(* Logix 5000 project; controller R5_CSS vendor 1 type 14 code 74 rev 19.11; software revision 19.01; part 9 of 20 *)
(* tags used below, declared in another part *)
   AC102A_BLEED_MAKEUP_STATUS : DINT;   // 0=stopped 1=bleed water 2=makeup water 3=wait
   AC102A_BLEED_START_TON : TIMER;
   AlarmMaster : DINT;
   F1_LC302 : LEVEL_CONTROL;
   F1_LC303A : LEVEL_CONTROL;
   F1_LC370 : LEVEL_CONTROL;
   FC365_LC370_FLOW_AUTO_SP : REAL;
   FC365_MAX_TIME_MIN : DINT;
   FC370 : FLOW_CONTROL;   // COALESCER MAKE UP WATER FLOW CONTROL
   FC370_FEED_ALARM_DISABLE : BOOL;
   FireFlowAlarmFromUTL : BOOL;
   LC302 : LEVEL_CONTROL;   // COALESCER OIL CHAMBER LEVEL CONTROL
   LC303 : LEVEL_CONTROL;   // COALESCER DIFFEENCE BETWEEN INTERFACE AND AQUEOUS PHASE
   LC303A : LEVEL_CONTROL;   // AQUEOUS PHASE OF PRIMARY SETTLER
   LC303B : LEVEL_CONTROL;   // INTERFACE LEVEL OF PRIMARY CONDENSER
   LC304 : LEVEL_CONTROL;   // SETTLER SECONDARY TANK INTERFACE LEVEL
   LC365_AUTO_SP_START : REAL;
   LC370 : LEVEL_CONTROL;   // WATER MAKE UP FOR PRIMARY SETTLER
   LC370_AUTO_ONS1 : BOOL;
   LC370_AUTO_ONS2 : BOOL;
   LC370_AUTO_SP_START : REAL;
   LC370_Bleed_Makeup_Started : BOOL;
   LC370_FLOW_TOO_LONG_ALM : BOOL;
   LC370_FLOW_TOO_LONG_RESETPB : BOOL;
   LC370_FLOW_TOO_LONG_TMR : TIMER;
   LC370_HMI_MAKEUP_ENABLE : BOOL;
   LC370_HMI_MAKEUP_REQ : BOOL;
   LC370_HMI_MAKEUP_START_ENABLE : BOOL;
   LC370_HMI_MAKEUP_START_PB : BOOL;
   LC370_HMI_MAKEUP_STOP_PB : BOOL;
   LC370_MAKEUP_AUTO_START_TON : TIMER;
   LC370_MANUAL_ONS1 : BOOL;
   LC370_Started : BOOL;
   LC370_TOTAl_GAL : REAL;
   LC370_TOTAl_RESET : BOOL;
   LC370_TOTAl_RESET_PB : BOOL;
   LC370_TOTALIZE : Totalize;
   LC370_TOTALIZE_EN : BOOL;
   LC370_UNABLE_TO_MAKEUP : BOOL;
   PID_LC370_Enable : BOOL;
   PID_LC370_Enable_ONS : BOOL;
   PID_LC370_Enable_Ton : TIMER;
   PID_LCV370 : PID;
   PID_LCV370_TON : TIMER;
   TC313A : TEMP_CONTROL;   // PRIMARY COALESCER SEPARATOR TEMPERATURE CONTROL
   TMR_FAULT : DINT;
(* MainProgram, continued *)

ROUTINE LC302_CoalOilChamberLevel   (* ladder *)
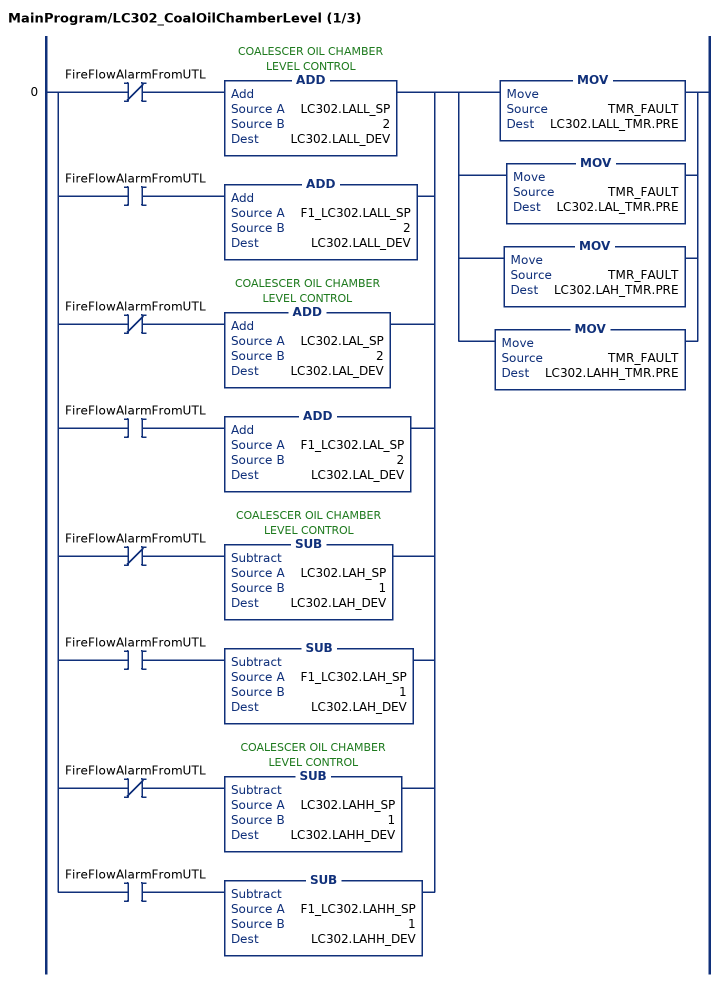
   0: [[XIO(FireFlowAlarmFromUTL) ADD(LC302.LALL_SP,2,LC302.LALL_DEV) ,XIC(FireFlowAlarmFromUTL) ADD(F1_LC302.LALL_SP,2,LC302.LALL_DEV) ] ,[XIO(FireFlowAlarmFromUTL) ADD(LC302.LAL_SP,2,LC302.LAL_DEV) ,XIC(FireFlowAlarmFromUTL) ADD(F1_LC302.LAL_SP,2,LC302.LAL_DEV) ] ,[XIO(FireFlowAlarmFromUTL) SUB(LC302.LAH_SP,1,LC302.LAH_DEV) ,XIC(FireFlowAlarmFromUTL) SUB(F1_LC302.LAH_SP,1,LC302.LAH_DEV) ] ,[XIO(FireFlowAlarmFromUTL) SUB(LC302.LAHH_SP,1,LC302.LAHH_DEV) ,XIC(FireFlowAlarmFromUTL) SUB(F1_LC302.LAHH_SP,1,LC302.LAHH_DEV) ] ][MOV(TMR_FAULT,LC302.LALL_TMR.PRE) ,MOV(TMR_FAULT,LC302.LAL_TMR.PRE) ,MOV(TMR_FAULT,LC302.LAH_TMR.PRE) ,MOV(TMR_FAULT,LC302.LAHH_TMR.PRE) ];
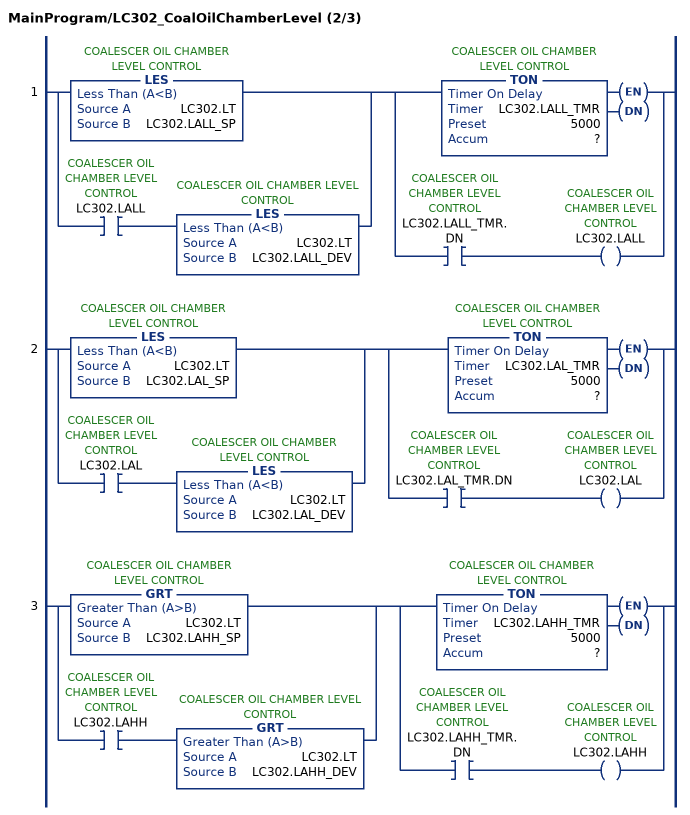
   1: [LES(LC302.LT,LC302.LALL_SP) ,XIC(LC302.LALL) LES(LC302.LT,LC302.LALL_DEV) ][TON(LC302.LALL_TMR,?,?) ,XIC(LC302.LALL_TMR.DN) OTE(LC302.LALL) ];
   2: [LES(LC302.LT,LC302.LAL_SP) ,XIC(LC302.LAL) LES(LC302.LT,LC302.LAL_DEV) ][TON(LC302.LAL_TMR,?,?) ,XIC(LC302.LAL_TMR.DN) OTE(LC302.LAL) ];
   3: [GRT(LC302.LT,LC302.LAHH_SP) ,XIC(LC302.LAHH) GRT(LC302.LT,LC302.LAHH_DEV) ][TON(LC302.LAHH_TMR,?,?) ,XIC(LC302.LAHH_TMR.DN) OTE(LC302.LAHH) ];
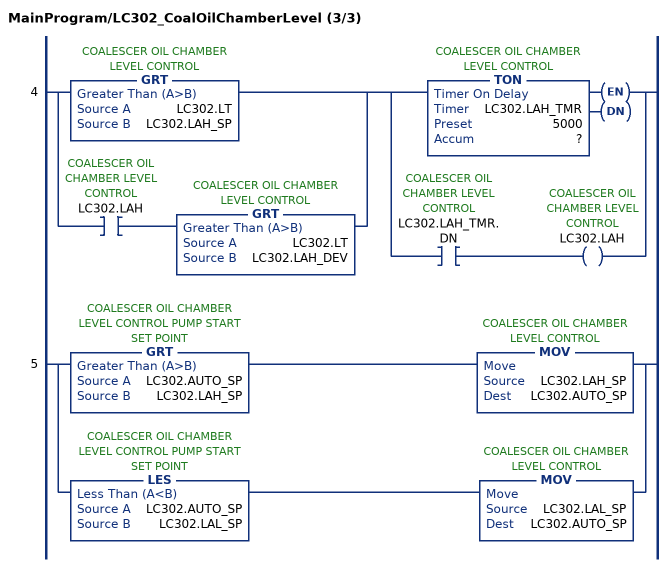
   4: [GRT(LC302.LT,LC302.LAH_SP) ,XIC(LC302.LAH) GRT(LC302.LT,LC302.LAH_DEV) ][TON(LC302.LAH_TMR,?,?) ,XIC(LC302.LAH_TMR.DN) OTE(LC302.LAH) ];
   5: [GRT(LC302.AUTO_SP,LC302.LAH_SP) MOV(LC302.LAH_SP,LC302.AUTO_SP) ,LES(LC302.AUTO_SP,LC302.LAL_SP) MOV(LC302.LAL_SP,LC302.AUTO_SP) ];
END_ROUTINE

ROUTINE LC303_CoalPriChamberInterfaceDiff   (* ladder *)
// LEVEL DIFFERENTIAL COALESCER TANK
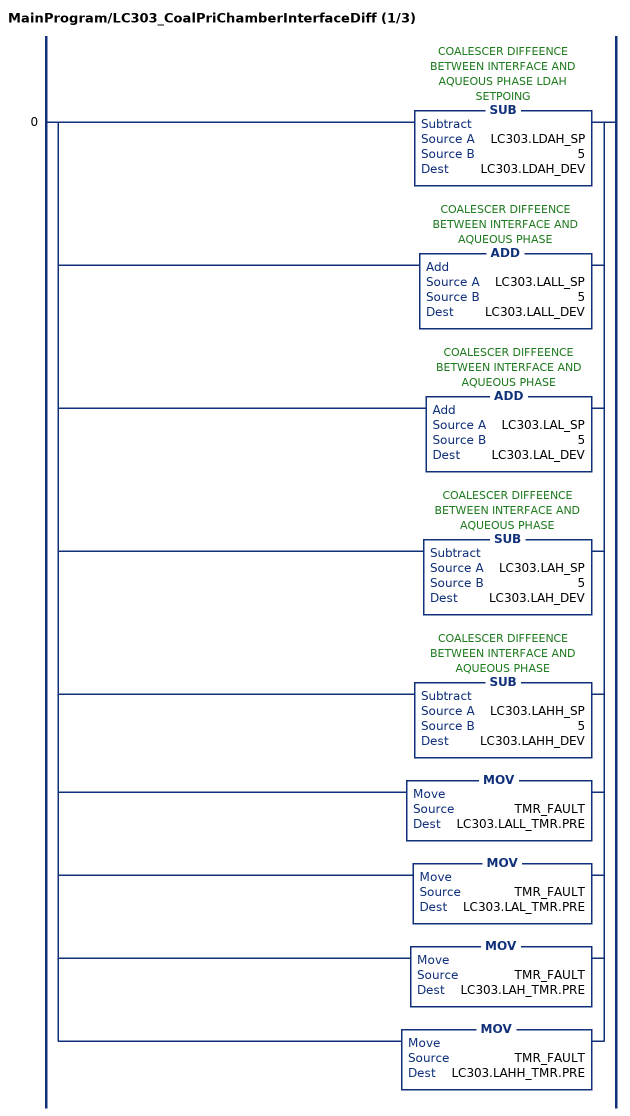
   0: [SUB(LC303.LDAH_SP,5,LC303.LDAH_DEV) ,ADD(LC303.LALL_SP,5,LC303.LALL_DEV) ,ADD(LC303.LAL_SP,5,LC303.LAL_DEV) ,SUB(LC303.LAH_SP,5,LC303.LAH_DEV) ,SUB(LC303.LAHH_SP,5,LC303.LAHH_DEV) ,MOV(TMR_FAULT,LC303.LALL_TMR.PRE) ,MOV(TMR_FAULT,LC303.LAL_TMR.PRE) ,MOV(TMR_FAULT,LC303.LAH_TMR.PRE) ,MOV(TMR_FAULT,LC303.LAHH_TMR.PRE) ];
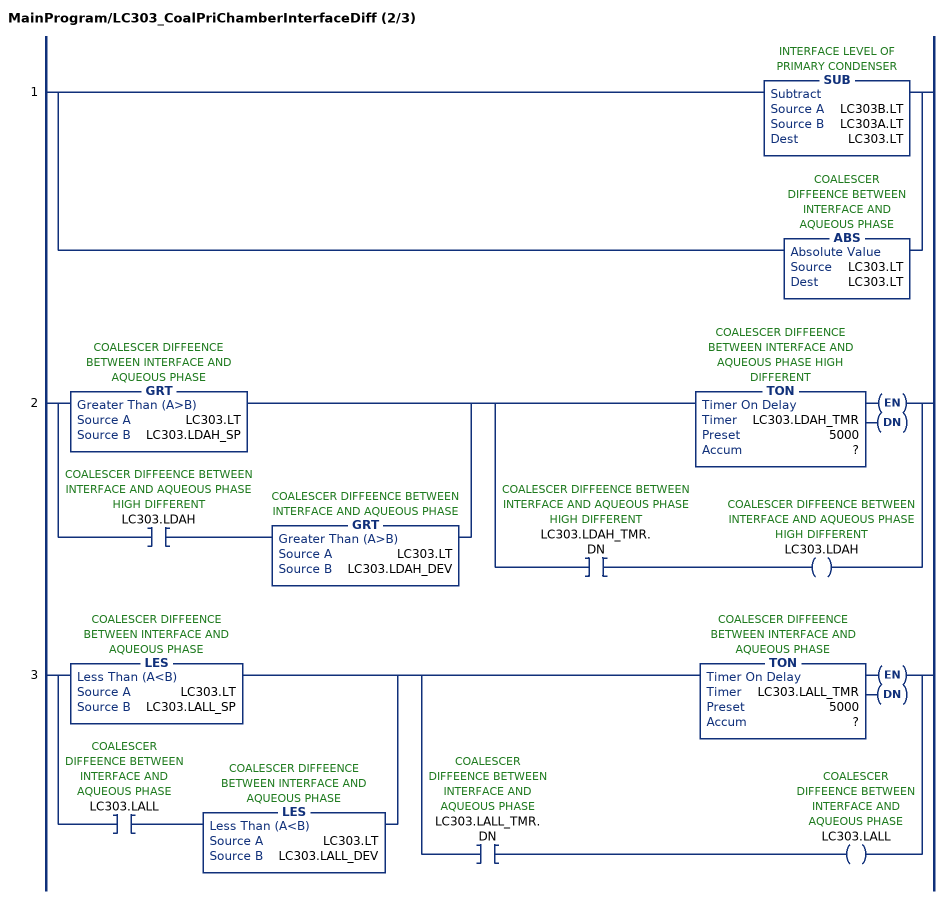
   1: [SUB(LC303B.LT,LC303A.LT,LC303.LT) ,ABS(LC303.LT,LC303.LT) ];
   2: [GRT(LC303.LT,LC303.LDAH_SP) ,XIC(LC303.LDAH) GRT(LC303.LT,LC303.LDAH_DEV) ][TON(LC303.LDAH_TMR,?,?) ,XIC(LC303.LDAH_TMR.DN) OTE(LC303.LDAH) ];
   3: [LES(LC303.LT,LC303.LALL_SP) ,XIC(LC303.LALL) LES(LC303.LT,LC303.LALL_DEV) ][TON(LC303.LALL_TMR,?,?) ,XIC(LC303.LALL_TMR.DN) OTE(LC303.LALL) ];
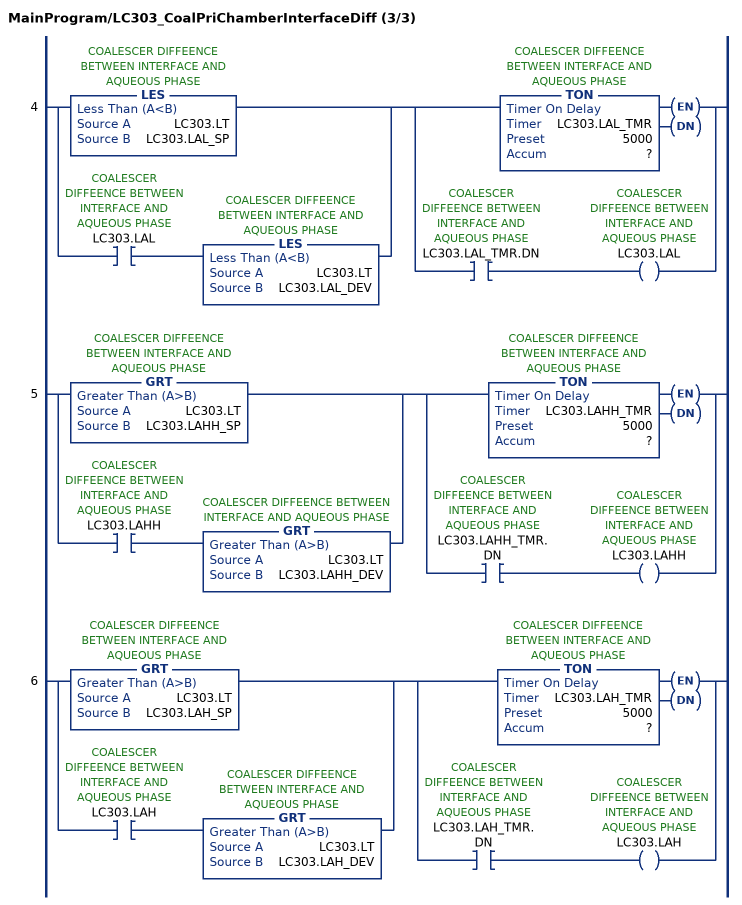
   4: [LES(LC303.LT,LC303.LAL_SP) ,XIC(LC303.LAL) LES(LC303.LT,LC303.LAL_DEV) ][TON(LC303.LAL_TMR,?,?) ,XIC(LC303.LAL_TMR.DN) OTE(LC303.LAL) ];
   5: [GRT(LC303.LT,LC303.LAHH_SP) ,XIC(LC303.LAHH) GRT(LC303.LT,LC303.LAHH_DEV) ][TON(LC303.LAHH_TMR,?,?) ,XIC(LC303.LAHH_TMR.DN) OTE(LC303.LAHH) ];
   6: [GRT(LC303.LT,LC303.LAH_SP) ,XIC(LC303.LAH) GRT(LC303.LT,LC303.LAH_DEV) ][TON(LC303.LAH_TMR,?,?) ,XIC(LC303.LAH_TMR.DN) OTE(LC303.LAH) ];
END_ROUTINE

ROUTINE LC303A_CoalPriChamberTopOfWater   (* ladder *)
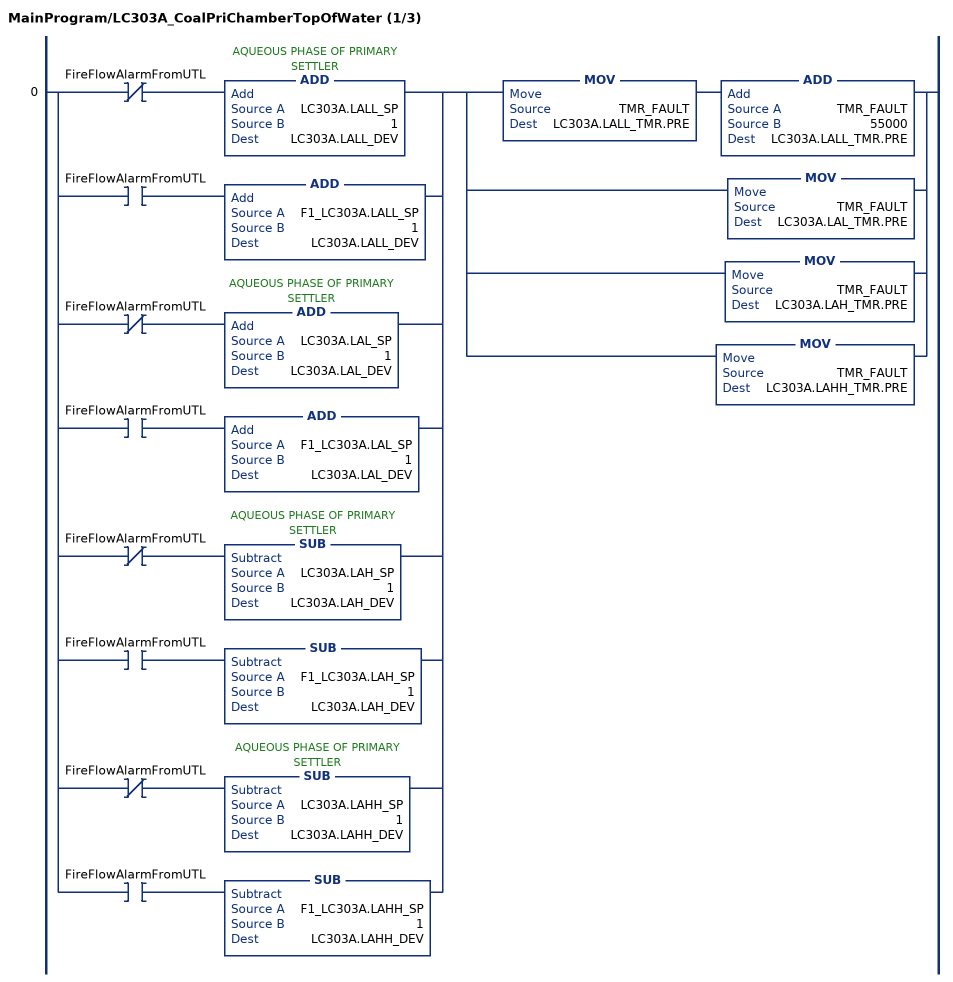
   0: [[XIO(FireFlowAlarmFromUTL) ADD(LC303A.LALL_SP,1,LC303A.LALL_DEV) ,XIC(FireFlowAlarmFromUTL) ADD(F1_LC303A.LALL_SP,1,LC303A.LALL_DEV) ] ,[XIO(FireFlowAlarmFromUTL) ADD(LC303A.LAL_SP,1,LC303A.LAL_DEV) ,XIC(FireFlowAlarmFromUTL) ADD(F1_LC303A.LAL_SP,1,LC303A.LAL_DEV) ] ,[XIO(FireFlowAlarmFromUTL) SUB(LC303A.LAH_SP,1,LC303A.LAH_DEV) ,XIC(FireFlowAlarmFromUTL) SUB(F1_LC303A.LAH_SP,1,LC303A.LAH_DEV) ] ,[XIO(FireFlowAlarmFromUTL) SUB(LC303A.LAHH_SP,1,LC303A.LAHH_DEV) ,XIC(FireFlowAlarmFromUTL) SUB(F1_LC303A.LAHH_SP,1,LC303A.LAHH_DEV) ] ][MOV(TMR_FAULT,LC303A.LALL_TMR.PRE) ADD(TMR_FAULT,55000,LC303A.LALL_TMR.PRE) ,MOV(TMR_FAULT,LC303A.LAL_TMR.PRE) ,MOV(TMR_FAULT,LC303A.LAH_TMR.PRE) ,MOV(TMR_FAULT,LC303A.LAHH_TMR.PRE) ];
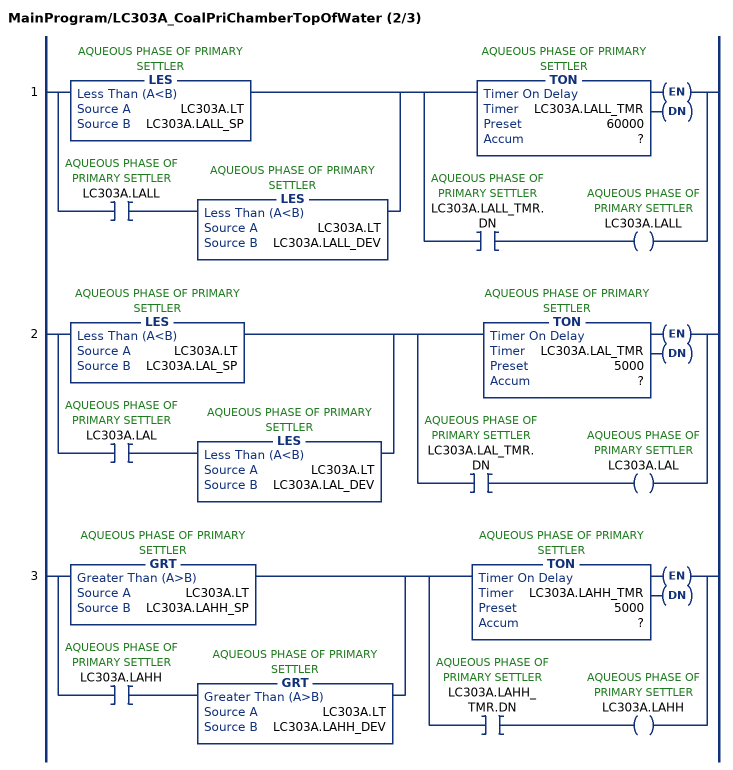
   1: [LES(LC303A.LT,LC303A.LALL_SP) ,XIC(LC303A.LALL) LES(LC303A.LT,LC303A.LALL_DEV) ][TON(LC303A.LALL_TMR,?,?) ,XIC(LC303A.LALL_TMR.DN) OTE(LC303A.LALL) ];
   2: [LES(LC303A.LT,LC303A.LAL_SP) ,XIC(LC303A.LAL) LES(LC303A.LT,LC303A.LAL_DEV) ][TON(LC303A.LAL_TMR,?,?) ,XIC(LC303A.LAL_TMR.DN) OTE(LC303A.LAL) ];
   3: [GRT(LC303A.LT,LC303A.LAHH_SP) ,XIC(LC303A.LAHH) GRT(LC303A.LT,LC303A.LAHH_DEV) ][TON(LC303A.LAHH_TMR,?,?) ,XIC(LC303A.LAHH_TMR.DN) OTE(LC303A.LAHH) ];
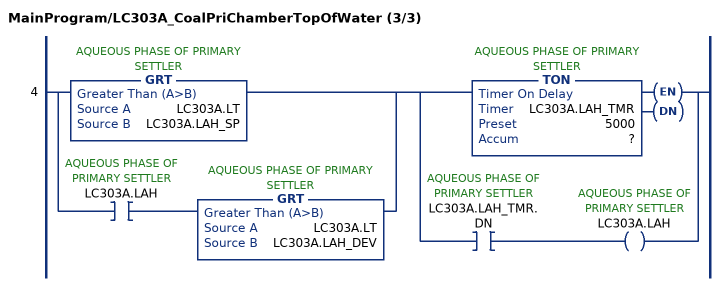
   4: [GRT(LC303A.LT,LC303A.LAH_SP) ,XIC(LC303A.LAH) GRT(LC303A.LT,LC303A.LAH_DEV) ][TON(LC303A.LAH_TMR,?,?) ,XIC(LC303A.LAH_TMR.DN) OTE(LC303A.LAH) ];
END_ROUTINE

ROUTINE LC303B_CoalPriChamberBottomOfOil   (* ladder *)
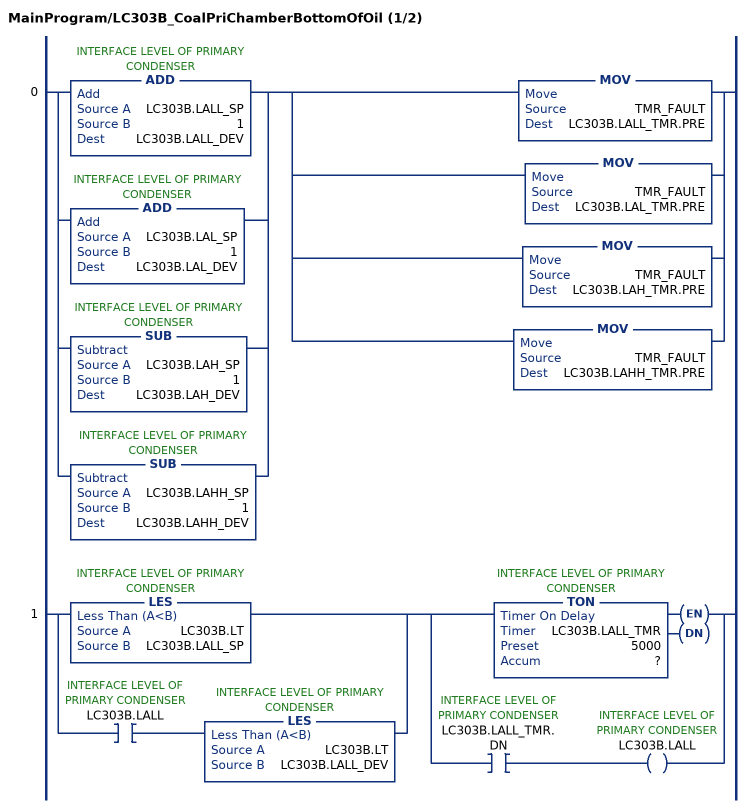
   0: [ADD(LC303B.LALL_SP,1,LC303B.LALL_DEV) ,ADD(LC303B.LAL_SP,1,LC303B.LAL_DEV) ,SUB(LC303B.LAH_SP,1,LC303B.LAH_DEV) ,SUB(LC303B.LAHH_SP,1,LC303B.LAHH_DEV) ][MOV(TMR_FAULT,LC303B.LALL_TMR.PRE) ,MOV(TMR_FAULT,LC303B.LAL_TMR.PRE) ,MOV(TMR_FAULT,LC303B.LAH_TMR.PRE) ,MOV(TMR_FAULT,LC303B.LAHH_TMR.PRE) ];
   1: [LES(LC303B.LT,LC303B.LALL_SP) ,XIC(LC303B.LALL) LES(LC303B.LT,LC303B.LALL_DEV) ][TON(LC303B.LALL_TMR,?,?) ,XIC(LC303B.LALL_TMR.DN) OTE(LC303B.LALL) ];
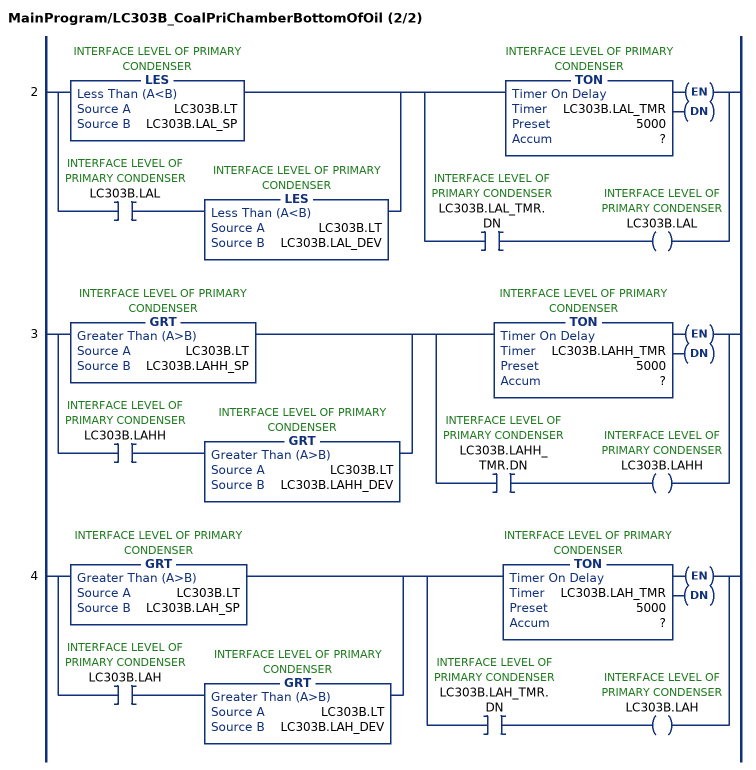
   2: [LES(LC303B.LT,LC303B.LAL_SP) ,XIC(LC303B.LAL) LES(LC303B.LT,LC303B.LAL_DEV) ][TON(LC303B.LAL_TMR,?,?) ,XIC(LC303B.LAL_TMR.DN) OTE(LC303B.LAL) ];
   3: [GRT(LC303B.LT,LC303B.LAHH_SP) ,XIC(LC303B.LAHH) GRT(LC303B.LT,LC303B.LAHH_DEV) ][TON(LC303B.LAHH_TMR,?,?) ,XIC(LC303B.LAHH_TMR.DN) OTE(LC303B.LAHH) ];
   4: [GRT(LC303B.LT,LC303B.LAH_SP) ,XIC(LC303B.LAH) GRT(LC303B.LT,LC303B.LAH_DEV) ][TON(LC303B.LAH_TMR,?,?) ,XIC(LC303B.LAH_TMR.DN) OTE(LC303B.LAH) ];
END_ROUTINE

ROUTINE LC304A_CoalSecChamberTopOfWater   (* ladder *)
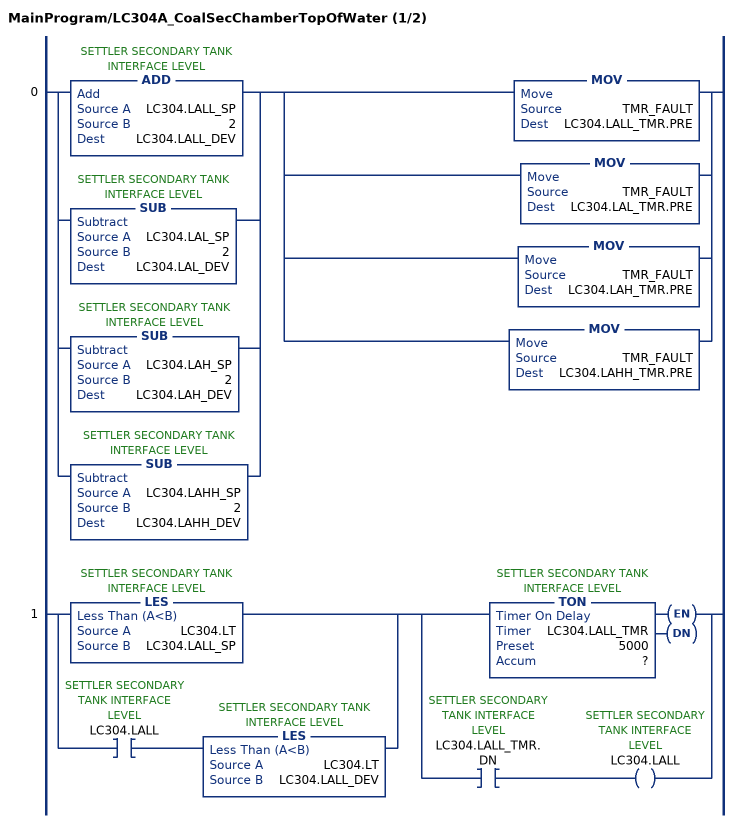
   0: [ADD(LC304.LALL_SP,2,LC304.LALL_DEV) ,SUB(LC304.LAL_SP,2,LC304.LAL_DEV) ,SUB(LC304.LAH_SP,2,LC304.LAH_DEV) ,SUB(LC304.LAHH_SP,2,LC304.LAHH_DEV) ][MOV(TMR_FAULT,LC304.LALL_TMR.PRE) ,MOV(TMR_FAULT,LC304.LAL_TMR.PRE) ,MOV(TMR_FAULT,LC304.LAH_TMR.PRE) ,MOV(TMR_FAULT,LC304.LAHH_TMR.PRE) ];
   1: [LES(LC304.LT,LC304.LALL_SP) ,XIC(LC304.LALL) LES(LC304.LT,LC304.LALL_DEV) ][TON(LC304.LALL_TMR,?,?) ,XIC(LC304.LALL_TMR.DN) OTE(LC304.LALL) ];
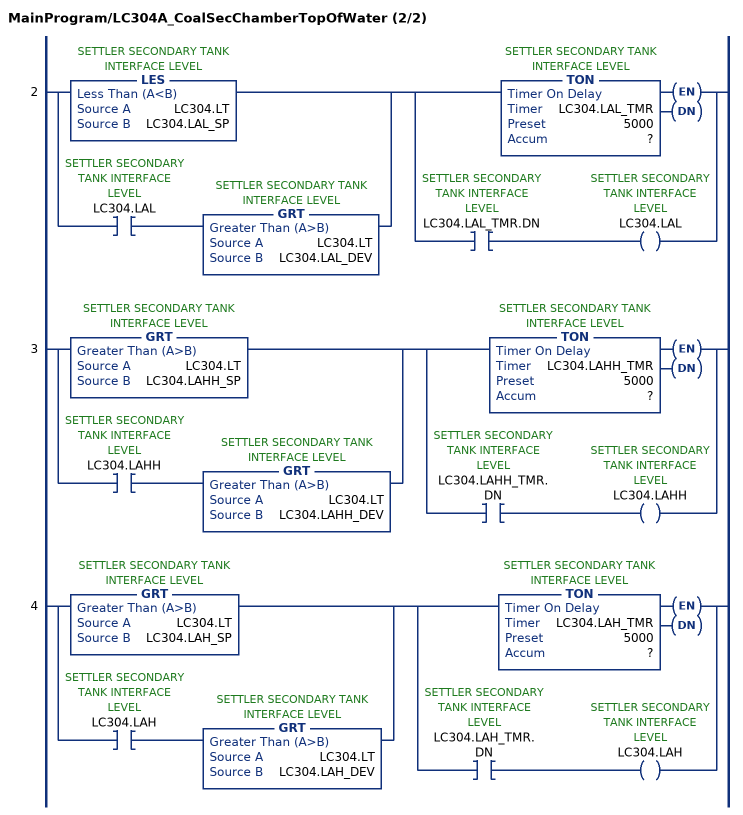
   2: [LES(LC304.LT,LC304.LAL_SP) ,XIC(LC304.LAL) GRT(LC304.LT,LC304.LAL_DEV) ][TON(LC304.LAL_TMR,?,?) ,XIC(LC304.LAL_TMR.DN) OTE(LC304.LAL) ];
   3: [GRT(LC304.LT,LC304.LAHH_SP) ,XIC(LC304.LAHH) GRT(LC304.LT,LC304.LAHH_DEV) ][TON(LC304.LAHH_TMR,?,?) ,XIC(LC304.LAHH_TMR.DN) OTE(LC304.LAHH) ];
   4: [GRT(LC304.LT,LC304.LAH_SP) ,XIC(LC304.LAH) GRT(LC304.LT,LC304.LAH_DEV) ][TON(LC304.LAH_TMR,?,?) ,XIC(LC304.LAH_TMR.DN) OTE(LC304.LAH) ];
END_ROUTINE

ROUTINE LC370_WaterMakeupLevel_PID   (* ladder *)
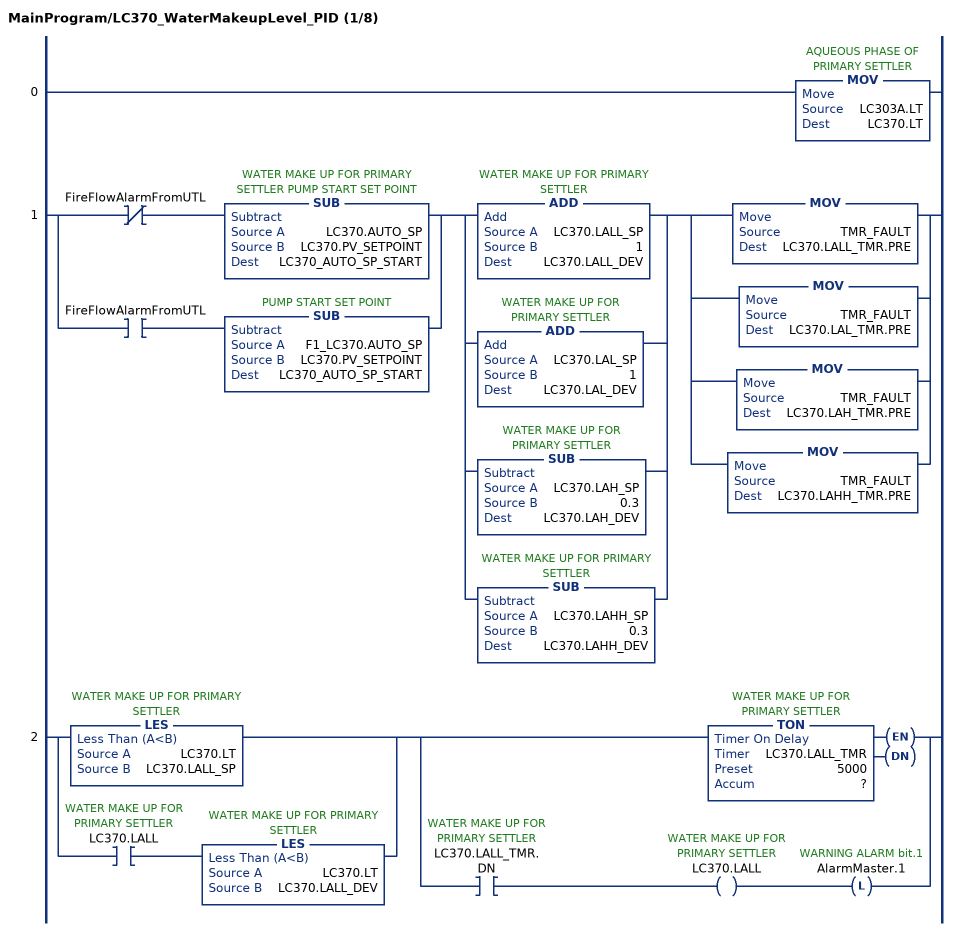
   0: MOV(LC303A.LT,LC370.LT);
   1: [XIO(FireFlowAlarmFromUTL) SUB(LC370.AUTO_SP,LC370.PV_SETPOINT,LC370_AUTO_SP_START) ,XIC(FireFlowAlarmFromUTL) SUB(F1_LC370.AUTO_SP,LC370.PV_SETPOINT,LC370_AUTO_SP_START) ][ADD(LC370.LALL_SP,1,LC370.LALL_DEV) ,ADD(LC370.LAL_SP,1,LC370.LAL_DEV) ,SUB(LC370.LAH_SP,0.3,LC370.LAH_DEV) ,SUB(LC370.LAHH_SP,0.3,LC370.LAHH_DEV) ][MOV(TMR_FAULT,LC370.LALL_TMR.PRE) ,MOV(TMR_FAULT,LC370.LAL_TMR.PRE) ,MOV(TMR_FAULT,LC370.LAH_TMR.PRE) ,MOV(TMR_FAULT,LC370.LAHH_TMR.PRE) ];
   2: [LES(LC370.LT,LC370.LALL_SP) ,XIC(LC370.LALL) LES(LC370.LT,LC370.LALL_DEV) ][TON(LC370.LALL_TMR,?,?) ,XIC(LC370.LALL_TMR.DN) OTE(LC370.LALL) OTL(AlarmMaster.1) ];
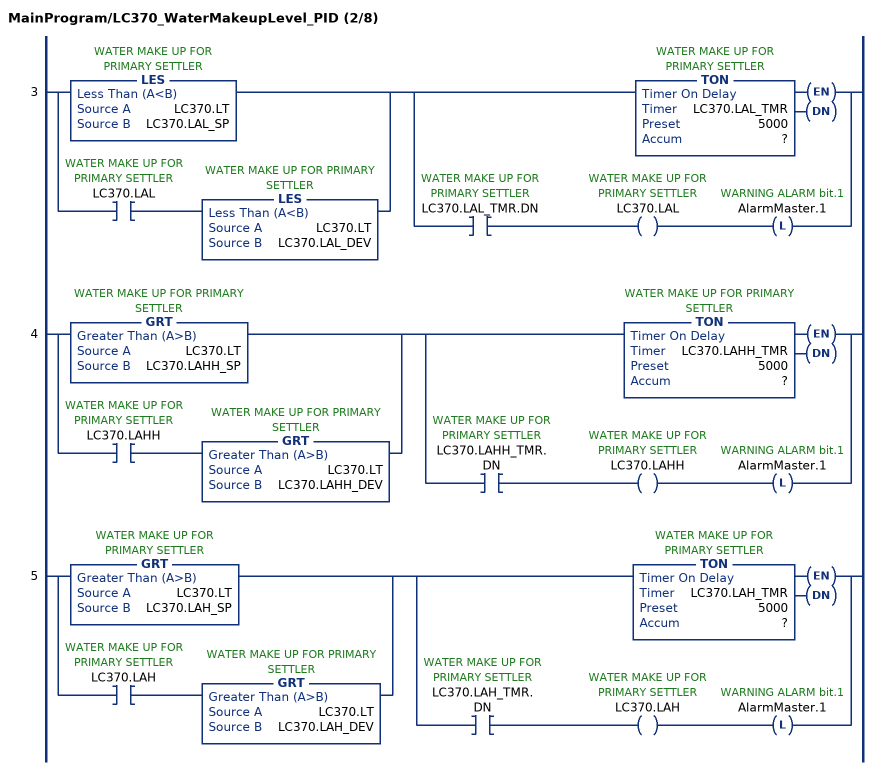
   3: [LES(LC370.LT,LC370.LAL_SP) ,XIC(LC370.LAL) LES(LC370.LT,LC370.LAL_DEV) ][TON(LC370.LAL_TMR,?,?) ,XIC(LC370.LAL_TMR.DN) OTE(LC370.LAL) OTL(AlarmMaster.1) ];
   4: [GRT(LC370.LT,LC370.LAHH_SP) ,XIC(LC370.LAHH) GRT(LC370.LT,LC370.LAHH_DEV) ][TON(LC370.LAHH_TMR,?,?) ,XIC(LC370.LAHH_TMR.DN) OTE(LC370.LAHH) OTL(AlarmMaster.1) ];
   5: [GRT(LC370.LT,LC370.LAH_SP) ,XIC(LC370.LAH) GRT(LC370.LT,LC370.LAH_DEV) ][TON(LC370.LAH_TMR,?,?) ,XIC(LC370.LAH_TMR.DN) OTE(LC370.LAH) OTL(AlarmMaster.1) ];
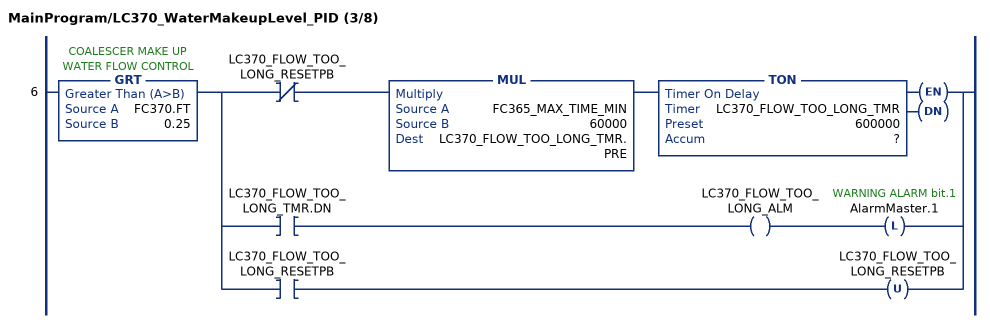
   6: GRT(FC370.FT,0.25)[XIO(LC370_FLOW_TOO_LONG_RESETPB) MUL(FC365_MAX_TIME_MIN,60000,LC370_FLOW_TOO_LONG_TMR.PRE) TON(LC370_FLOW_TOO_LONG_TMR,?,?) ,XIC(LC370_FLOW_TOO_LONG_TMR.DN) OTE(LC370_FLOW_TOO_LONG_ALM) OTL(AlarmMaster.1) ,XIC(LC370_FLOW_TOO_LONG_RESETPB) OTU(LC370_FLOW_TOO_LONG_RESETPB) ];
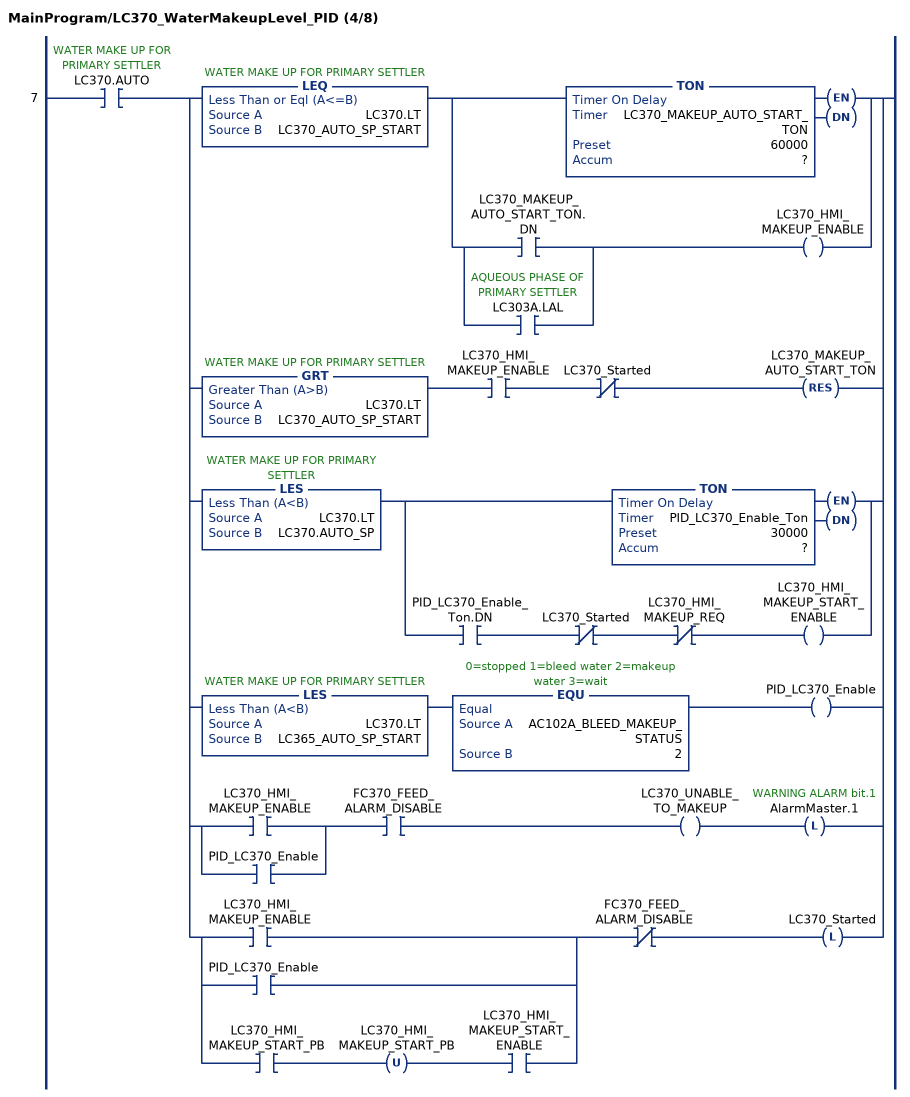
   7: XIC(LC370.AUTO)[LEQ(LC370.LT,LC370_AUTO_SP_START) [TON(LC370_MAKEUP_AUTO_START_TON,?,?) ,[XIC(LC370_MAKEUP_AUTO_START_TON.DN) ,XIC(LC303A.LAL) ] OTE(LC370_HMI_MAKEUP_ENABLE) ] ,GRT(LC370.LT,LC370_AUTO_SP_START) XIC(LC370_HMI_MAKEUP_ENABLE) XIO(LC370_Started) RES(LC370_MAKEUP_AUTO_START_TON) ,LES(LC370.LT,LC370.AUTO_SP) [TON(PID_LC370_Enable_Ton,?,?) ,XIC(PID_LC370_Enable_Ton.DN) XIO(LC370_Started) XIO(LC370_HMI_MAKEUP_REQ) OTE(LC370_HMI_MAKEUP_START_ENABLE) ] ,LES(LC370.LT,LC365_AUTO_SP_START) EQU(AC102A_BLEED_MAKEUP_STATUS,2) OTE(PID_LC370_Enable) ,[XIC(LC370_HMI_MAKEUP_ENABLE) ,XIC(PID_LC370_Enable) ] XIC(FC370_FEED_ALARM_DISABLE) OTE(LC370_UNABLE_TO_MAKEUP) OTL(AlarmMaster.1) ,[XIC(LC370_HMI_MAKEUP_ENABLE) ,XIC(PID_LC370_Enable) ,XIC(LC370_HMI_MAKEUP_START_PB) OTU(LC370_HMI_MAKEUP_START_PB) XIC(LC370_HMI_MAKEUP_START_ENABLE) ] XIO(FC370_FEED_ALARM_DISABLE) OTL(LC370_Started) ];
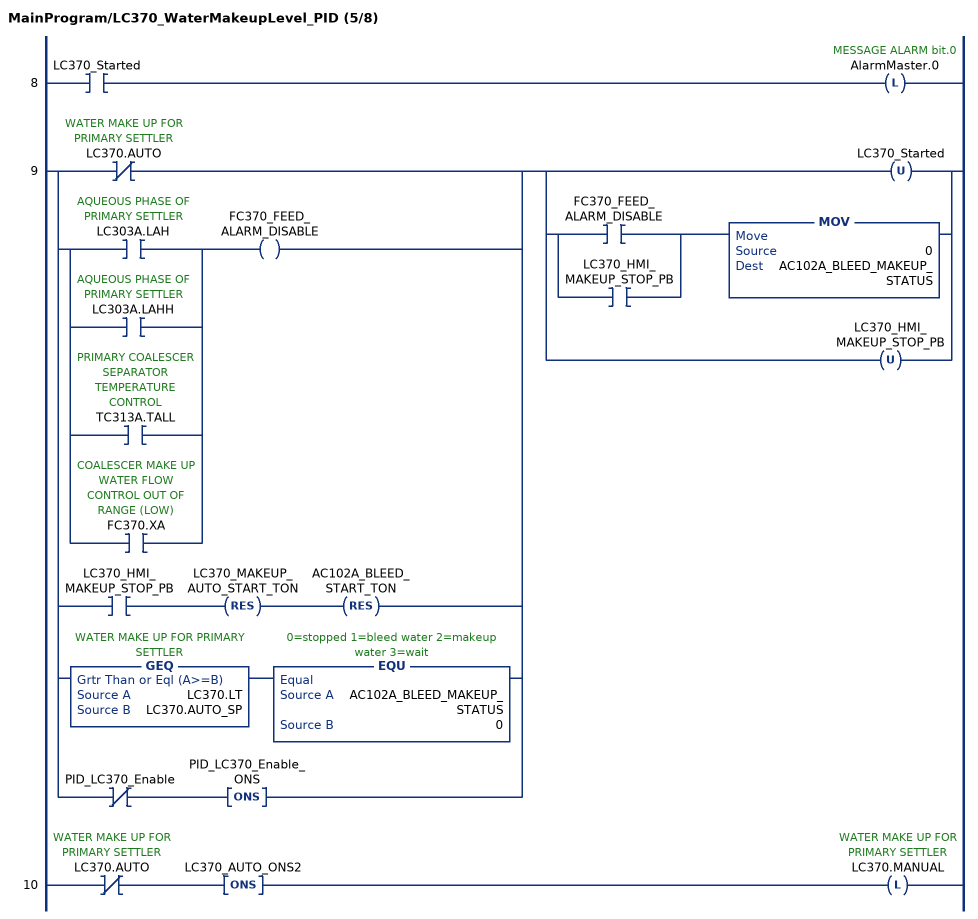
   8: XIC(LC370_Started)OTL(AlarmMaster.0);
   9: [XIO(LC370.AUTO) ,[XIC(LC303A.LAH) ,XIC(LC303A.LAHH) ,XIC(TC313A.TALL) ,XIC(FC370.XA) ] OTE(FC370_FEED_ALARM_DISABLE) ,XIC(LC370_HMI_MAKEUP_STOP_PB) RES(LC370_MAKEUP_AUTO_START_TON) RES(AC102A_BLEED_START_TON) ,GEQ(LC370.LT,LC370.AUTO_SP) EQU(AC102A_BLEED_MAKEUP_STATUS,0) ,XIO(PID_LC370_Enable) ONS(PID_LC370_Enable_ONS) ][OTU(LC370_Started) ,[XIC(FC370_FEED_ALARM_DISABLE) ,XIC(LC370_HMI_MAKEUP_STOP_PB) ] MOV(0,AC102A_BLEED_MAKEUP_STATUS) ,OTU(LC370_HMI_MAKEUP_STOP_PB) ];
   10: XIO(LC370.AUTO)ONS(LC370_AUTO_ONS2)OTL(LC370.MANUAL);
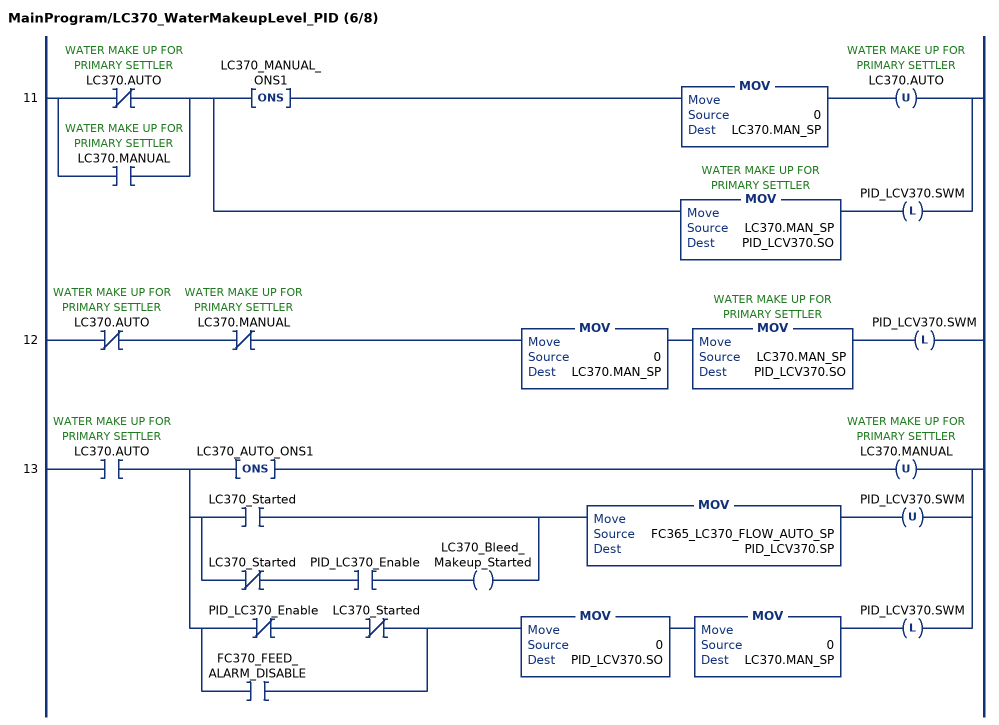
   11: [XIO(LC370.AUTO) ,XIC(LC370.MANUAL) ][ONS(LC370_MANUAL_ONS1) MOV(0,LC370.MAN_SP) OTU(LC370.AUTO) ,MOV(LC370.MAN_SP,PID_LCV370.SO) OTL(PID_LCV370.SWM) ];
   12: XIO(LC370.AUTO)XIO(LC370.MANUAL)MOV(0,LC370.MAN_SP)MOV(LC370.MAN_SP,PID_LCV370.SO)OTL(PID_LCV370.SWM);
   13: XIC(LC370.AUTO)[ONS(LC370_AUTO_ONS1) OTU(LC370.MANUAL) ,[XIC(LC370_Started) ,XIO(LC370_Started) XIC(PID_LC370_Enable) OTE(LC370_Bleed_Makeup_Started) ] MOV(FC365_LC370_FLOW_AUTO_SP,PID_LCV370.SP) OTU(PID_LCV370.SWM) ,[XIO(PID_LC370_Enable) XIO(LC370_Started) ,XIC(FC370_FEED_ALARM_DISABLE) ] MOV(0,PID_LCV370.SO) MOV(0,LC370.MAN_SP) OTL(PID_LCV370.SWM) ];
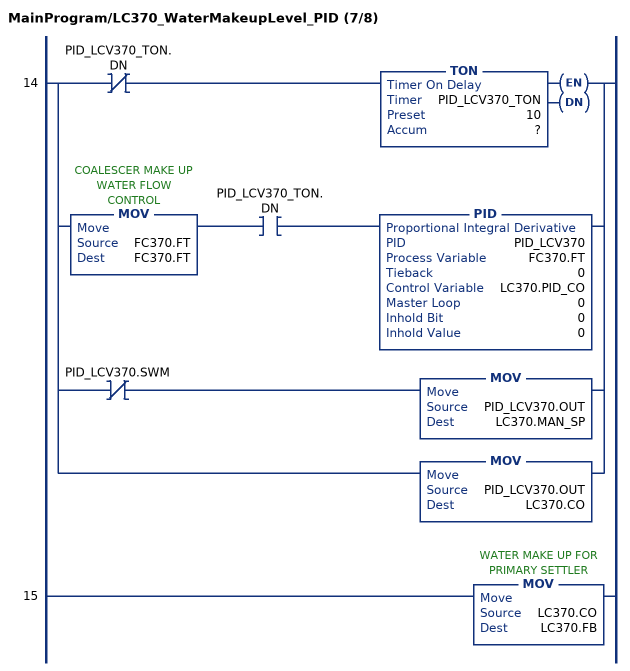
   14: [XIO(PID_LCV370_TON.DN) TON(PID_LCV370_TON,?,?) ,MOV(FC370.FT,FC370.FT) XIC(PID_LCV370_TON.DN) PID(PID_LCV370,FC370.FT,0,LC370.PID_CO,0,0,0) ,XIO(PID_LCV370.SWM) MOV(PID_LCV370.OUT,LC370.MAN_SP) ,MOV(PID_LCV370.OUT,LC370.CO) ];
   15: MOV(LC370.CO,LC370.FB);
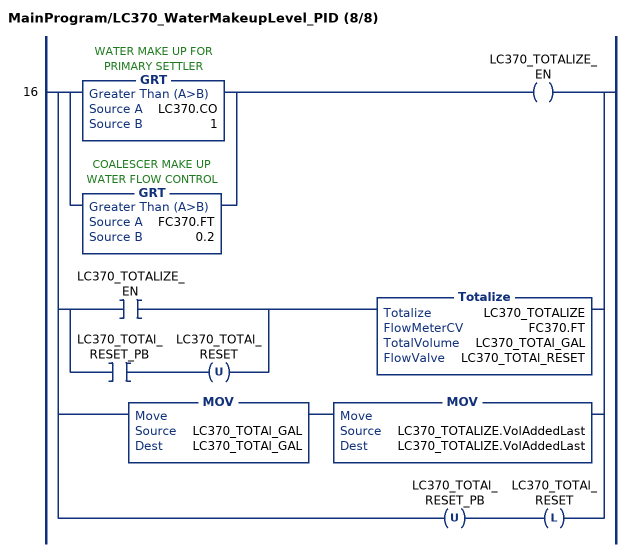
   16: [[GRT(LC370.CO,1) ,GRT(FC370.FT,0.2) ] OTE(LC370_TOTALIZE_EN) ,[XIC(LC370_TOTALIZE_EN) ,XIC(LC370_TOTAl_RESET_PB) OTU(LC370_TOTAl_RESET) ] Totalize(LC370_TOTALIZE,FC370.FT,LC370_TOTAl_GAL,LC370_TOTAl_RESET) ,MOV(LC370_TOTAl_GAL,LC370_TOTAl_GAL) MOV(LC370_TOTALIZE.VolAddedLast,LC370_TOTALIZE.VolAddedLast) ,OTU(LC370_TOTAl_RESET_PB) OTL(LC370_TOTAl_RESET) ];
END_ROUTINE
